# EPICS IOC start-up script: iocsh/ethercatmcDctEL1252-PILS.iocsh
dbLoadRecords("ethercatmcDctEL1252-PILS.template", "PREFIX=$(PREFIX), MOTOR_PORT=$(MOTOR_PORT)")
